TYPE ST_OpStates :
STRUCT
	Selected			: BOOL;
	Ready				: BOOL;
	Start				: BOOL;
	Stop				: BOOL;
	Reset				: BOOL;
END_STRUCT
END_TYPE

(* stored: Version 1.1.0.1, ProductVersion 3.1.0.19
   DUT ST_OpStates: Id {0d4dd5bf-38f5-4fb4-884e-24c9014c566d} *)
